// TIA Portal project "S7-1500 ile Sayıcı ile 3 Motor Kontrolü" (V18)

(* hardware
DEVICE "S7-1500/ET200MP station_1"  S7-1500 station
   slot 0: "Rail_0"  Rack  6ES7 590-1***0-0AA0
   slot 1: "PLC_1"  CPU 1512C-1 PN  6ES7 512-1CK01-0AB0  V2.8
      slot 3: "CPU display_1"  6ES7591-1AA00-0AA0
      slot 32768: "PROFINET interface_1"  X1
         slot 32769: "Port_1"  X1 P1
         slot 32770: "Port_2"  X1 P2
      slot 34817: "Virtual CP interface port_1"  Virtual CP interface port  Virtual CP interface port
DEVICE "HMI_1"  KTP700 Basic PN
   slot 0: "HMI_1"  KTP700 Basic PN  6AV2 123-2GB03-0AX0  14.0.1.0
   slot 1: "HMI_RT_1"  KTP700 Basic PN  6AV2 123-2GB03-0AX0  14.0.1.0
   slot 5: "HMI_1.IE_CP_1"  PROFINET Interface  14.0.1.0
      slot 1: "PROFINET Interface_1"  PROFINET Interface
         slot 1: "Port_1"  Port
*)

// ===== PLC "PLC_1"  CPU 1512C-1 PN =====

VAR_GLOBAL   // PLC tag table "Default tag table"
   "Stop" AT %M0.0 : Bool;
   "Start" AT %M0.1 : Bool;
   "Sayıcı İçeriği" AT %MW100 : Int;
   "1. Motor" AT %Q0.0 : Bool;
   "2. Motor" AT %Q0.1 : Bool;
   "3. Motor" AT %Q0.2 : Bool;
END_VAR

// folder: System blocks/Program resources

DATA_BLOCK "IEC_Counter_0_DB"   // DB1
{ S7_Optimized_Access := 'TRUE' }
AUTHOR : Simatic
FAMILY : IEC
NAME : CNTR
VERSION : 1.0
// stored: InstanceOfName IEC_COUNTER
"IEC_COUNTER"
BEGIN
END_DATA_BLOCK

// folder: (top level)

ORGANIZATION_BLOCK "Main"   // OB1, LAD, ProgramCycle
TITLE = "Main Program Sweep (Cycle)"
{ S7_Optimized_Access := 'TRUE' }
VERSION : 0.1
   VAR_INPUT
      Initial_Call : Bool;   // Initial call of this OB
      Remanence : Bool;   // =True, if remanent data are available
   END_VAR
   VAR_TEMP   // added for the SCL form of the ladder/FBD networks
      _w1 : Bool;
   END_VAR
BEGIN

REGION Network 1: Sayıcı ile Motor Kontrolü
   // Starta;
   // 1. basışta 1. motor
   // 2. basışta 2. motor
   // 3. basışta 3. motor
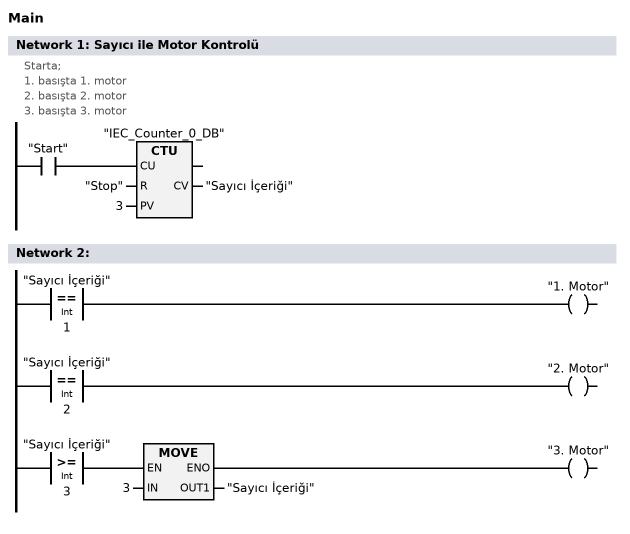
   "IEC_Counter_0_DB".CTU(CU := "Start", R := "Stop", PV := 3, CV => "Sayıcı İçeriği");
END_REGION

REGION Network 2
   RUNG wire#powerrail
      { S7_Templates := "SrcType := Int" } EQ_Contact(in1 := "Sayıcı İçeriği", in2 := 1)
      Coil( "1. Motor" )
   END_RUNG
   RUNG wire#powerrail
      { S7_Templates := "SrcType := Int" } EQ_Contact(in1 := "Sayıcı İçeriği", in2 := 2)
      Coil( "2. Motor" )
   END_RUNG
   RUNG wire#powerrail
      { S7_Templates := "SrcType := Int" } GE_Contact(in1 := "Sayıcı İçeriği", in2 := 3)
      Move(in := 3, out1 => "Sayıcı İçeriği")
      Coil( "3. Motor" )
   END_RUNG
   // the same network as SCL:
   "1. Motor" := "Sayıcı İçeriği" = 1;
   "2. Motor" := "Sayıcı İçeriği" = 2;
   #_w1 := "Sayıcı İçeriği" >= 3;
   IF #_w1 THEN "Sayıcı İçeriği" := 3; END_IF;
   "3. Motor" := #_w1;
END_REGION
END_ORGANIZATION_BLOCK

(* ===== HMI "HMI_RT_1" =====
system functions are stored by id; their names below are inferred from use
connection "Connection_1": ETHERNET, SMART_S7_1500_OMS
connection "HMI_Connection_1": ETHERNET, SMART_S7_1500_OMS

HMI tags "Default tag table"
   "Sayıcı İçeriği" : Int = PLC "Sayıcı İçeriği" AT %MW100, 100 ms
   "Stop" : Bool = PLC Stop AT %M0.0, 100 ms
   "Start" : Bool = PLC Start AT %M0.1, 100 ms
   "3. Motor" : Bool = PLC "3. Motor" AT %Q0.2, 100 ms
   "2. Motor" : Bool = PLC "2. Motor" AT %Q0.1, 100 ms
   "1. Motor" : Bool = PLC "1. Motor" AT %Q0.0, 100 ms
   "Tag_ScreenNumber" : Int = PLC "Sayıcı İçeriği" AT %MW100, 100 ms

graphic list "Geri Hareket": 0 'Graphic_22'; 1 'Graphic_23'

graphic list "İleri Hareket": 0 'Graphic_21'; 1 'Graphic_20'

Template "Template_1" 800x480
   Button "Exit" at 714,429 size 71x50; TextOff 'Exit'; PictureOff "ExitRuntime_KTP700_Basic_PN_TR"; PictureOn "ExitRuntime_KTP700_Basic_PN_TR"
      on Release: StopRuntime(0)
   Button "Language" at 614,429 size 71x50; TextOff 'Language'; PictureOff "ToggleLanguage_KTP700_Basic_PN_TR"; PictureOn "ToggleLanguage_KTP700_Basic_PN_TR"
      on Release: function_fb9197e8(-1)
   Button "Log on" at 514,429 size 71x50; TextOff 'Log on'; PictureOff "Login_KTP700_Basic_PN_TR"; PictureOn "Login_KTP700_Basic_PN_TR"
      on Release: function_a2a04561()
   Button "Alarms" at 114,429 size 71x50; TextOff 'Alarms'; PictureOff "AlarmDisplay_KTP700_Basic_PN_TR"; PictureOn "AlarmDisplay_KTP700_Basic_PN_TR"
      on Release: function_ef3f5d25("Alarm window_Unacknowledged", -1)
   Button "Start screen" at 14,429 size 71x50; TextOff 'Start screen'; PictureOff "NavigateHome_KTP700_Basic_PN_TR"; PictureOn "NavigateHome_KTP700_Basic_PN_TR"
      on Release: ActivateScreen("Root screen", 0)
   SymbolicIOField "Symbolic_IO_Field_Screen" at 93,9 size 600x33; TextOff '0'; TextOn '1'; TextList "TextList_ScreenNames"
      on Change: ActivateScreenByNumber("Sayıcı İçeriği", 0)
      ProcessValue <- "Tag_ScreenNumber"
   DateTimeField "HmiScreenItemData" at 695,25 size 105x25
   DateTimeField "HmiScreenItemData_1" at 695,0 size 105x25
   GraphicView "Logo" at 0,0 size 91x51; Picture "Logo of HMI_1"

screen "Root screen" 800x480, template "Template_1"
   on GenerateScreen: SetTag("Tag_ScreenNumber", 1)
   Button "Button_4" at 409,131 size 129x50; TextOff 'Start'
      on Press: InvertBit("Start")
      on Release: ResetBit("Start")
   Circle "Circle_1" at 316,93 size 52x52
      Appearance <- "1. Motor"
   Circle "Circle_2" at 316,214 size 52x52
      Appearance <- "3. Motor"
   Circle "Circle_3" at 316,154 size 52x52
      Appearance <- "2. Motor"
   Button "Button_1" at 409,198 size 129x50; TextOff 'Stop'
      on Press: SetBit("Stop")
      on Release: ResetBit("Stop")
   IOField "I/O field_1" at 280,301 size 129x54; FormatPattern s9999999999
      ProcessValue <- "Sayıcı İçeriği"
   TextField "Text field_1" at 129,113 size 16x23; Text 'Text'
   TextField "Text field_2" at 207,236 size 73x23; Text '3. Motor'
   TextField "Text field_3" at 207,170 size 68x23; Text '2.Motor'
   TextField "Text field_4" at 207,113 size 68x23; Text '1.Motor'
*)